(* IEC 61131-3 sources: learning-path/04_introduction_to_st/exercises/2_implement_tank/src, 2 files *)

(* ---- configuration.st ---- *)
USING Siemens.AxTraining.ControlModules;
USING Siemens.AxTraining;

CONFIGURATION PLC_1
    TASK Main(Interval := T#10ms, Priority := 1);
    PROGRAM P1 WITH Main: FluidProgram;

    VAR_GLOBAL
        ctrlOpenInletValve : BOOL;
        inletValve : Valve;
    END_VAR
END_CONFIGURATION

(* ---- fluidProgram.st ---- *)
USING Siemens.AxTraining.ControlModules;

NAMESPACE Siemens.AxTraining
    PROGRAM FluidProgram

        VAR_EXTERNAL
            ctrlOpenInletValve : BOOL;
            inletValve : Valve;
        END_VAR

        inletValve(ctrlOpen => ctrlOpenInletValve);
    END_PROGRAM
END_NAMESPACE
